FUNCTION_BLOCK FB_AbsorptionChiller
VAR_INPUT
END_VAR
VAR_OUTPUT
END_VAR
VAR
END_VAR

END_FUNCTION_BLOCK

(* stored: Version 1.1.0.1, ProductVersion 3.1.4024.10
   POU FB_AbsorptionChiller: Id {58c6b46c-a56b-418c-b518-17d466272f79}, SpecialFunc None *)
